{attribute 'linkalways'} 
{attribute 'no_explicit_call' := 'This FB is a CLASS and must be accessed using methods or properties'}
{attribute 'enable_dynamic_creation'}
FUNCTION_BLOCK FINAL MAX_BYTE EXTENDS Node
VAR
	in1 : _BYTE(0);
	in2 : _BYTE(0);
	out : _BYTE(0);
END_VAR

METHOD PUBLIC Clone : I_Node
VAR
	pNode : POINTER TO MAX_BYTE;
END_VAR
pNode := __NEW(MAX_BYTE);
Clone := pNode^;
END_METHOD

METHOD FB_init : BOOL
VAR_INPUT
	bInitRetains : BOOL; // if TRUE, the retain variables are initialized (warm start / cold start)
	bInCopyCode : BOOL;  // if TRUE, the instance afterwards gets moved into the copy code (online change)
END_VAR
AddInput('in1',THIS^.in1);
AddInput('in2',THIS^.in2);
AddOutput('out', THIS^.out);
END_METHOD

METHOD PROTECTED OnExecute
VAR
END_VAR
out.Value := MAX(in1.Value, in2.Value);
END_METHOD

END_FUNCTION_BLOCK

(* stored: Version 1.1.0.1, ProductVersion 3.1.4024.15
   POU MAX_BYTE: Id {7cd17e1f-39bc-467e-bf31-1120643ef104}, SpecialFunc None
   Folder Constructor: Id {82e9cd34-868a-4416-9374-f165f65e6ad6}
   Method Clone: Id {0fe8d4d4-ab2d-4f6d-90f9-6d1711acf1e0}
   Method FB_init: Id {a206408f-ac06-48ae-9796-06b38b3cfa44}
   Method OnExecute: Id {e675eeef-d5ac-4c8f-8001-0f8d0f8f104f} *)
